// TIA Portal V19 export
ORGANIZATION_BLOCK "Main"   // OB1, LAD, ProgramCycle
TITLE = "Main Program Sweep (Cycle)"
{ S7_Optimized_Access := 'TRUE' }
// stored: SetENOAutomatically false
   VAR_INPUT
      Initial_Call : Bool;   // Initial call of this OB
      Remanence : Bool;   // =True, if remanent data are available
   END_VAR
BEGIN

REGION Network 1
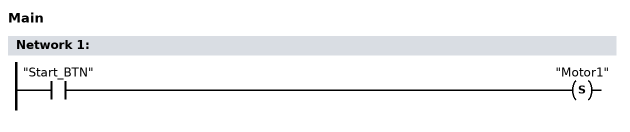
   RUNG wire#powerrail
      Contact( "Start_BTN" )
      S_Coil( "Motor1" )
   END_RUNG
   // the same network as SCL:
   IF "Start_BTN" THEN "Motor1" := TRUE; END_IF;
END_REGION
END_ORGANIZATION_BLOCK
